// TwinCAT 3 PLC project MotionController
// ProgramVersion: 3.1.4020.4
// libraries:
//   LCLS Motion Control, * (SLAC)
//   LCLS General, * (SLAC)
//   Tc2_Standard, * (Beckhoff Automation GmbH)
//   Tc2_System, * (Beckhoff Automation GmbH)
//   Tc3_Module, * (Beckhoff Automation GmbH)
// project tree:
//   DUTs/ ST_BeamDemand.TcDUT, ST_MotorDriver.TcDUT, ST_BisscEncoder.TcDUT
//   GVLs/ SendBeamDemand.TcGVL
//   / PlcTask.TcTTO
//   POUs/ BisscEvaluator.TcPOU, count_mgr_test.TcPOU, MAIN.TcPOU
// real-time tasks:
//   TASK PlcTask: cycle T#10ms, priority 20, ADS port 350
// I/O:
//   DEVICE Device 1 (EtherCAT) (disabled), AmsNetId 134.79.86.210.2.1
//     Term 1 (EK1200) [EK1200-5000 EtherCAT Power supply (2A E-Bus)]
//       Term 2 (EL6695) [EL6695 EtherCAT Bridge terminal (Primary)]
// variable links:
//   HutchMPS Instance <-> MotionController/MotionController Instance
//     PlcTask Inputs/GetBeamDemand.beamRate <-> PlcTask Outputs/SendBeamDemand.beamRate

CONFIGURATION MotionController
    RESOURCE PLC ON TwinCAT3
        TASK PlcTask(INTERVAL := T#10ms, PRIORITY := 20);
        PROGRAM MAIN WITH PlcTask : MAIN;
    END_RESOURCE
END_CONFIGURATION

// ---- DUTs/ST_BeamDemand.TcDUT
TYPE ST_BeamDemand :
STRUCT
	// What beam rate is required from a device? (Probably units of frequency) 
	beamRate : LREAL;
	// Demand specifies if this demand is an emergency (True). Non-Demand is for non-emergencies
	demand : BOOL;
END_STRUCT
END_TYPE

// ---- DUTs/ST_MotorDriver.TcDUT
TYPE ST_MotorDriver :
STRUCT
END_STRUCT
END_TYPE

// ---- DUTs/ST_BisscEncoder.TcDUT
TYPE ST_BisscEncoder :
STRUCT
	// Inclusive limits on encoder position (checks for values exceeding this inclusive range)
	// These values are just guesses - no units yet - no actual data - CHANGE BEFORE USE
	ncLLimit :	ULINT := 0;
	ncULimit :	ULINT := 100;
	// Readback for linear encoder's position
	encLoc	AT %I*	:	ULINT;
END_STRUCT
END_TYPE

// ---- GVLs/SendBeamDemand.TcGVL
{attribute 'qualified_only'}
VAR_GLOBAL
	// What beam rate is required from a device? (Probably units of frequency) 
	beamRate	AT %Q*	: LREAL;
	// Demand specifies if this demand is an emergency (True). Non-Demand is for non-emergencies/Preemtive protection (synonomous). Sent to Hutch PLC.
	// demand : BOOL;
END_VAR

// ---- POUs/MAIN.TcPOU
PROGRAM MAIN
VAR
	Counter0Inc : DWORD := 1;
	Counter0Read : DWORD; 
	Counter0 : count_mgr_test;
	Encoder0Read : ULINT;
	Encoder0	:	ST_BisscEncoder;
	EncoderDemand0 : ST_BeamDemand;
END_VAR

Counter0(Increment:=Counter0Inc);
Counter0Read := Counter0.CurrentOut;
EncoderDemand0 := BisscEvaluator(Encoder0);

END_PROGRAM

// ---- POUs/count_mgr_test.TcPOU
FUNCTION_BLOCK count_mgr_test
VAR_INPUT
	Increment : DWORD;
END_VAR
VAR_OUTPUT
	CurrentOut : DWORD;
END_VAR
VAR
	UpperLimit : DWORD := 500;
END_VAR
VAR PERSISTENT
	CurrentVal : DWORD := 0;
END_VAR

IF CurrentVal >= UpperLimit THEN
	CurrentVal := 0;
ELSE
	CurrentVal := CurrentVal + Increment;
END_IF



CurrentOut := CurrentVal;

END_FUNCTION_BLOCK

// ---- POUs/BisscEvaluator.TcPOU
FUNCTION BisscEvaluator : ST_BeamDemand
VAR_INPUT
	encoder : ST_BisscEncoder;
END_VAR
VAR	
	readLoc: ULINT;
	newDemand : ST_BeamDemand;
END_VAR

readLoc := Encoder.encLoc;
IF readLoc <= Encoder.ncULimit THEN
	newDemand.demand := TRUE;
ELSE
	newDemand.demand := FALSE;
END_IF

IF readLoc <= Encoder.ncULimit THEN 
	newDemand.beamRate := 0;
ELSE
	newDemand.beamRate := 50;
END_IF

BisscEvaluator := newDemand;

END_FUNCTION
